TYPE SMD12LaserConfig EXTENDS DeviceConfiguration :
STRUCT
	SerialCommunication : SerialCommunication;
END_STRUCT
END_TYPE

(* stored: Version 1.1.0.1, ProductVersion 3.1.4024.4
   DUT SMD12LaserConfig: Id {702be717-1d60-485f-952c-b539cdb5211a} *)
